(* Logix 5000 project; controller cal1632 1756-L62 rev 16.20; software revision 16.05; part 55 of 61 *)
(* tags used below, declared in another part *)
   p29_param_tension_hi_limit : REAL;   // Parameter Tension High Limit
   p29r16_drive_ok : BOOL;   // Winder B Drive Enable E-Stop Clear and Own Drive Healthy
   param_pos_db : REAL;   // C: Turret Position Dead Band
   pb_jog_turret_rev : BOOL;   // HMI PB: Jog Turret Rev
   turret_in_wda_run_position : BOOL;   // Turret In Winder A Run Position
   turret_in_wdb_run_position : BOOL;   // Turret In Winder B Run Position
   turret_index_permissive : BOOL;   // Turret Index Permissive No Turret Drive Fault AND Neither Winder Requesting Run
   wb_run_position : REAL;   // Turret Winder B Run Position
   wb_run_position_high_limit : REAL;
   wb_run_position_low_limit : REAL;
   winder_accel_rate : REAL;
   winder_decel_rate : REAL;
   AFI : BOOL;
   FAULT : BOOL;
   p00_wac : Accumulator;   // Winder Accumulator
   p00_wac_position_pct : REAL;   // Winder Accumulator Carriage Position Filtered [% of Stroke]
   p01_recipe_active : recipe;
   p01r02_plc_scan_time_in_sec : REAL;
   p01r09 : routine;
   p01r09_pb_global_reset : BOOL;
   p01r09_request_line_jog : BOOL;
   p01r13_line_running : BOOL;
   p01r13_line_slow_ramp : BOOL;
   p01r13_permissive_drives : BOOL;
   p02_real_from_hmi : hmi_real;
   p25_ao_selected_speed : REAL;
   p25r09_mode_thread : BOOL;
   p25r09_pb_jog_fwd : BOOL;
   p25r09_pb_jog_rev : BOOL;
   p29_ai_wb_torque : REAL;
   p29_ai_wdr_lc : REAL;
   p29_ao_wdrb_selected_speed : REAL;
   p29_di_wa_brake : BOOL;
   p29_di_wa_motor : BOOL;
   p29_di_wb_brake : BOOL;
   p29_di_wb_motor : BOOL;
   p29_di_wdr_b_start : BOOL;
   p29_di_wdr_b_stop : BOOL;
   p29_di_wdr_index_fwd : BOOL;
   p29_di_wdr_jog : BOOL;
   p29_param_payout_torque : REAL;   // Winder Torque Limit During Accumulator Payout Line Running [%]
   p29_param_soak : REAL;
   p29_param_start_speed_factor : REAL;   // Winder Start Speed Fraction of Line Speed Before Tension is Established Shared by Winder A and B
   p29_param_tension_ok_band : REAL;   // Winder Tension Established Band Shared by Winder A and B [lbf]
   p29_param_wind_out_speed : REAL;   // Winder Wind Out Speed Winder Speed with the Line Stopped Empties the Accumulator [fpm]
   p29_param_wind_out_stop_pct : REAL;   // Winder Wind Out Stop When the Accumulator Reaches This Position [% of Stroke]
   p29_param_wind_out_torque : REAL;   // Winder Torque Limit During Wind Out Line Stopped [%]
   p29_param_winder_accel_rate : REAL;   // Winder Common Speed Ramp Default Accel Rate Applied Only if winder_accel_rate is Zero
   p29_param_winder_decel_rate : REAL;   // Winder Common Speed Ramp Default Decel Rate Applied Only if winder_decel_rate is Zero
   p29_param_winder_jog_speed : REAL;
   p29_wda_status_word : INT;
   p29_wda_vfd : ABB_PROTOCOL_VFD;
   p29_wdb_control_word : INT;
   p29_wdb_status_word : INT;
   p29_wdb_vfd : ABB_PROTOCOL_VFD;
   p29r01 : routine;
   p29r02_tension_dev_max : REAL;
   p29r02_tension_dev_min : REAL;
   p29r02_wb_calc_torque_ref : REAL;
   p29r09_torque_mode : BOOL;
   p29r09_winder_b_active : BOOL;
   p29r11_index_active : BOOL;
   p29r11_speed_offset : REAL;
   p29r15 : routine;
   p29r15_request_run : BOOL;
   p29r15_run_permissive : BOOL;
   p29r15_timer_fault : TIMER[10];
   p29r15_timer_warning : TIMER[4];
   p29r15_wdra_active : BOOL;
   p29r16 : routine;
   p29r16_accel_rate : REAL;
   p29r16_acel_decel_ramp : SYS_ACC_DEC_RAMP;   // Winder B Speed Setpoint Ramp
   p29r16_ao_torque : REAL;
   p29r16_const_torque_ref : REAL;
   p29r16_decel_rate : REAL;
   p29r16_fast_accel_rate : REAL;
   p29r16_fast_decel_rate : REAL;
   p29r16_index_start_torque : REAL;
   p29r16_jog_torque_ref : REAL;
   p29r16_ramped_setpoint : REAL;   // Winder B Ramped Speed Setpoint [fpm]
   p29r16_request_jog_fwd : BOOL;
   p29r16_request_run : BOOL;
   p29r16_request_thread_fwd : BOOL;
   p29r16_request_thread_rev : BOOL;
   p29r16_run_permissive : BOOL;
   p29r16_selected_speed : REAL;
   p29r16_selected_torque : REAL;
   p29r16_soak_active : BOOL;
   p29r16_speed_factor : REAL;   // Winder B Speed Factor Multiplier on the Ramped Setpoint
   p29r16_speed_setpoint : REAL;   // Winder B Speed Setpoint [fpm]
   p29r16_state : DINT;
   p29r16_stop_dwell : TIMER;   // Winder B Stop Dwell Holds the winder after the stop PB so the nip closes first
   p29r16_tension_ok : BOOL;
   p29r16_thread_torque_ref : REAL;
   p29r16_timer_fault : TIMER[10];
   p29r16_timer_warning : TIMER[4];
   p29r16_torque_acc_rate : REAL;
   p29r16_torque_boost_acc_rate : REAL;
   p29r16_torque_boost_dec_rate : REAL;
   p29r16_torque_boost_ref : REAL;
   p29r16_torque_boost_timer : TIMER;
   p29r16_torque_dec_rate : REAL;
   p29r16_torque_fast_acc_rate : REAL;
   p29r16_torque_fast_dec_rate : REAL;
   p29r16_torque_high_ref : REAL;
   p29r16_torque_low_ref : REAL;
   p29r16_torque_mode_acc_rate : REAL;
   p29r16_torque_mode_dec_rate : REAL;
   p29r16_torque_ramp : SYS_ACC_DEC_RAMP;
   p29r16_torque_soak_acc_rate : REAL;
   p29r16_torque_soak_dec_rate : REAL;
   p29r16_torque_start_timer : TIMER;
   p29r16_vfd_start_request : BOOL;
   p29r16_wdrb_accel_decel : SYS_ACC_DEC_RAMP;
   p29r16_wdrb_active : BOOL;
   p29r16_wdrb_ramped_speed : REAL;
   p29r16_zero_speed : BOOL;
   p29r20 : routine;
(* P29_Winder, continued *)

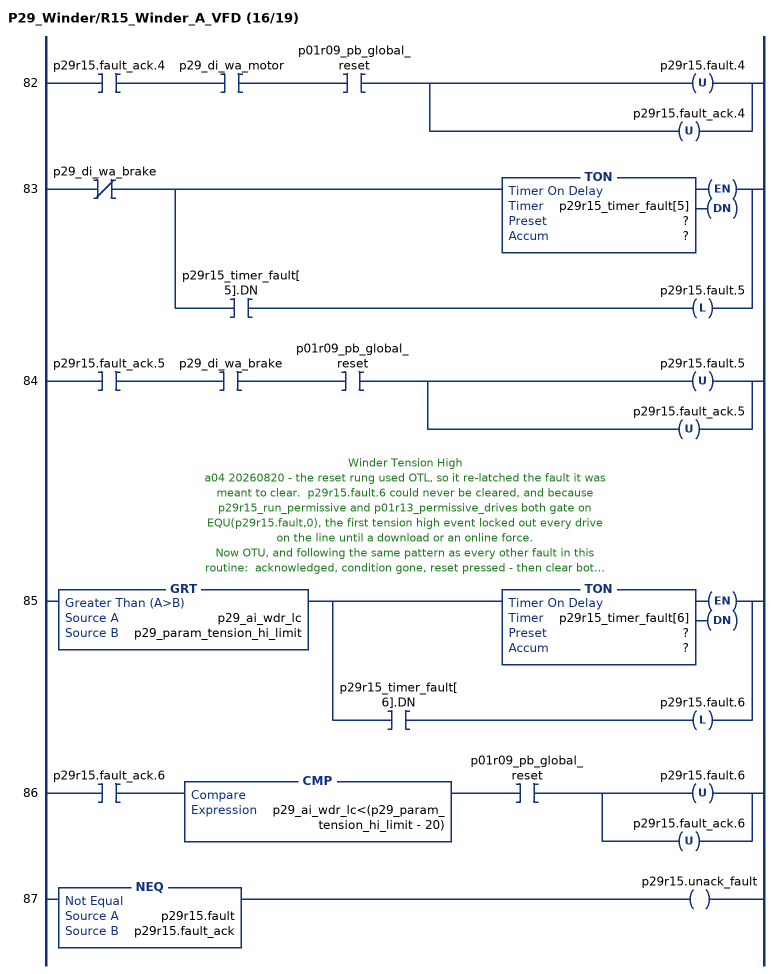
   [picture p1114: P29_Winder/R15_Winder_A_VFD rungs 82-87]
   82: XIC(p29r15.fault_ack.4)XIC(p29_di_wa_motor)XIC(p01r09_pb_global_reset)[OTU(p29r15.fault.4) ,OTU(p29r15.fault_ack.4) ];
   83: XIO(p29_di_wa_brake)[TON(p29r15_timer_fault[5],?,?) ,XIC(p29r15_timer_fault[5].DN) OTL(p29r15.fault.5) ];
   84: XIC(p29r15.fault_ack.5)XIC(p29_di_wa_brake)XIC(p01r09_pb_global_reset)[OTU(p29r15.fault.5) ,OTU(p29r15.fault_ack.5) ];
   // Winder Tension High
   // a04 20260820 - the reset rung used OTL, so it re-latched the fault it was
   // meant to clear.  p29r15.fault.6 could never be cleared, and because
   // p29r15_run_permissive and p01r13_permissive_drives both gate on
   // EQU(p29r15.fault,0), the first tension high event locked out every drive
   // on the line until a download or an online force.
   // Now OTU, and following the same pattern as every other fault in this
   // routine:  acknowledged, condition gone, reset pressed - then clear both
   // the fault bit and its ack bit so unack_fault clears with it.
   // Note p29_ai_wdr_lc is a single load cell shared by both winders, so a
   // tension excursion latches fault.6 on A and B together.  That is correct
   // for one web, but both need the reset.
   85: GRT(p29_ai_wdr_lc,p29_param_tension_hi_limit)[TON(p29r15_timer_fault[6],?,?) ,XIC(p29r15_timer_fault[6].DN) OTL(p29r15.fault.6) ];
   86: XIC(p29r15.fault_ack.6)CMP(p29_ai_wdr_lc<(p29_param_tension_hi_limit - 20))XIC(p01r09_pb_global_reset)[OTU(p29r15.fault.6) ,OTU(p29r15.fault_ack.6) ];
   87: NEQ(p29r15.fault,p29r15.fault_ack)OTE(p29r15.unack_fault);
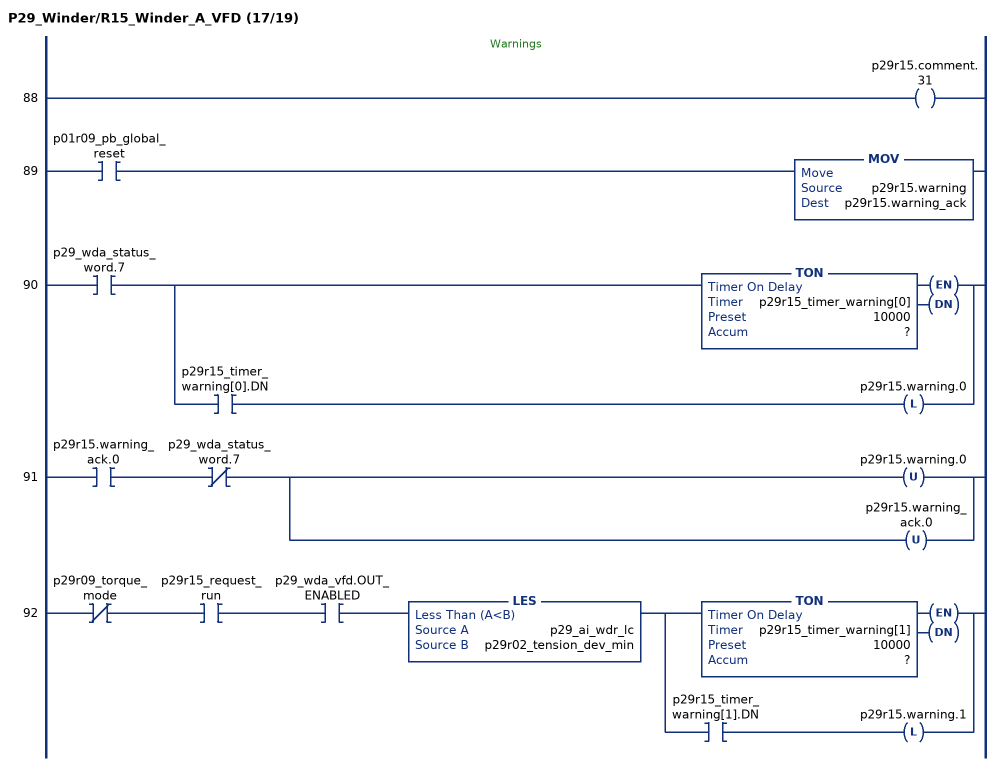
   // Warnings
   88: OTE(p29r15.comment.31);
   89: XIC(p01r09_pb_global_reset)MOV(p29r15.warning,p29r15.warning_ack);
   90: XIC(p29_wda_status_word.7)[TON(p29r15_timer_warning[0],?,?) ,XIC(p29r15_timer_warning[0].DN) OTL(p29r15.warning.0) ];
   91: XIC(p29r15.warning_ack.0)XIO(p29_wda_status_word.7)[OTU(p29r15.warning.0) ,OTU(p29r15.warning_ack.0) ];
   92: XIO(p29r09_torque_mode)XIC(p29r15_request_run)XIC(p29_wda_vfd.OUT_ENABLED)LES(p29_ai_wdr_lc,p29r02_tension_dev_min)[TON(p29r15_timer_warning[1],?,?) ,XIC(p29r15_timer_warning[1].DN) OTL(p29r15.warning.1) ];
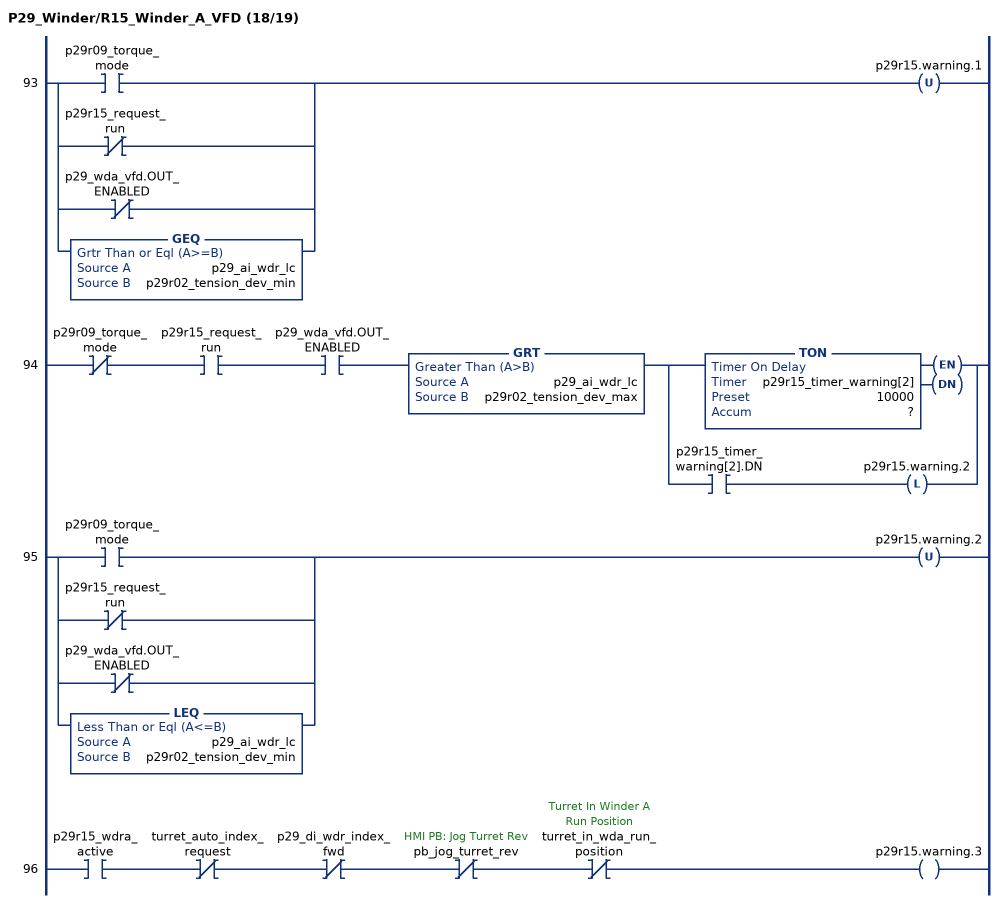
   93: [XIC(p29r09_torque_mode) ,XIO(p29r15_request_run) ,XIO(p29_wda_vfd.OUT_ENABLED) ,GEQ(p29_ai_wdr_lc,p29r02_tension_dev_min) ]OTU(p29r15.warning.1);
   94: XIO(p29r09_torque_mode)XIC(p29r15_request_run)XIC(p29_wda_vfd.OUT_ENABLED)GRT(p29_ai_wdr_lc,p29r02_tension_dev_max)[TON(p29r15_timer_warning[2],?,?) ,XIC(p29r15_timer_warning[2].DN) OTL(p29r15.warning.2) ];
   95: [XIC(p29r09_torque_mode) ,XIO(p29r15_request_run) ,XIO(p29_wda_vfd.OUT_ENABLED) ,LEQ(p29_ai_wdr_lc,p29r02_tension_dev_min) ]OTU(p29r15.warning.2);
   96: XIC(p29r15_wdra_active)XIO(turret_auto_index_request)XIO(p29_di_wdr_index_fwd)XIO(pb_jog_turret_rev)XIO(turret_in_wda_run_position)OTE(p29r15.warning.3);
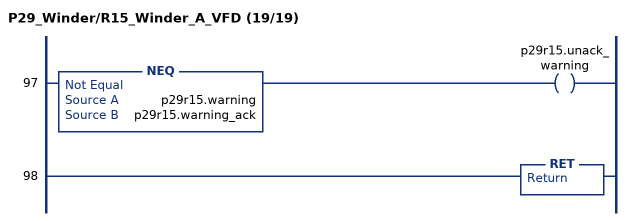
   97: NEQ(p29r15.warning,p29r15.warning_ack)OTE(p29r15.unack_warning);
   98: RET();
END_ROUTINE

ROUTINE R16_Winder_B_VFD   (* ladder *)
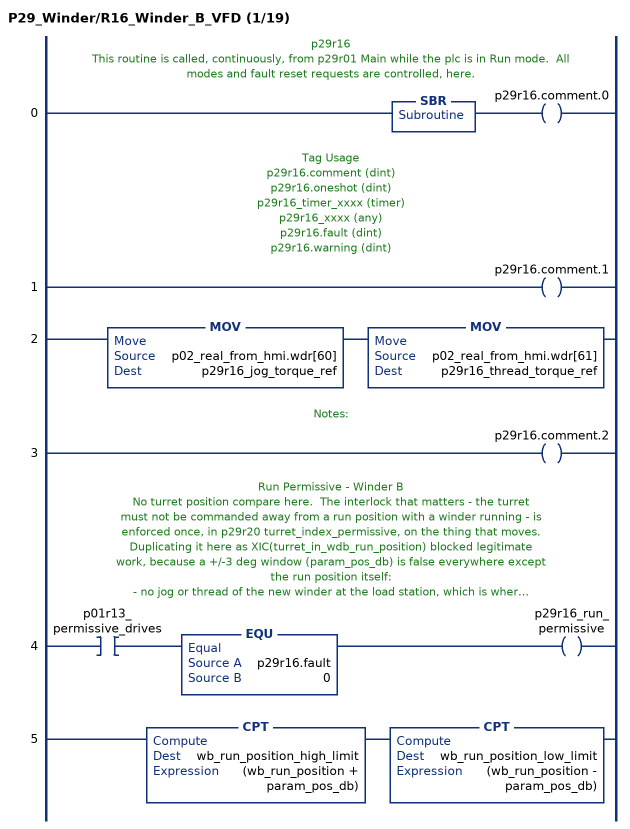
   // p29r16
   // This routine is called, continuously, from p29r01 Main while the plc is in Run mode.  All modes and fault reset requests are controlled, here.
   0: SBR()OTE(p29r16.comment.0);
   // Tag Usage
   // p29r16.comment (dint)
   // p29r16.oneshot (dint)
   // p29r16_timer_xxxx (timer)
   // p29r16_xxxx (any)
   // p29r16.fault (dint)
   // p29r16.warning (dint)
   1: OTE(p29r16.comment.1);
   2: MOV(p02_real_from_hmi.wdr[60],p29r16_jog_torque_ref)MOV(p02_real_from_hmi.wdr[61],p29r16_thread_torque_ref);
   // Notes:
   3: OTE(p29r16.comment.2);
   // Run Permissive - Winder B
   // No turret position compare here.  The interlock that matters - the turret
   // must not be commanded away from a run position with a winder running - is
   // enforced once, in p29r20 turret_index_permissive, on the thing that moves.
   // Duplicating it here as XIC(turret_in_wdb_run_position) blocked legitimate
   // work, because a +/-3 deg window (param_pos_db) is false everywhere except
   // the run position itself:
   //   - no jog or thread of the new winder at the load station, which is where
   //     the leader is attached and has to be wound on
   //   - no winding the tail off the doffed roll at doff position
   //   - no accumulator wind-out unless the turret happens to be at run
   //   - the winder dropped out 0.7 s into a doff index, web still tensioned
   // Rev 20260825 a23
   4: XIC(p01r13_permissive_drives)EQU(p29r16.fault,0)OTE(p29r16_run_permissive);
   5: CPT(wb_run_position_high_limit,(wb_run_position + param_pos_db))CPT(wb_run_position_low_limit,(wb_run_position - param_pos_db));
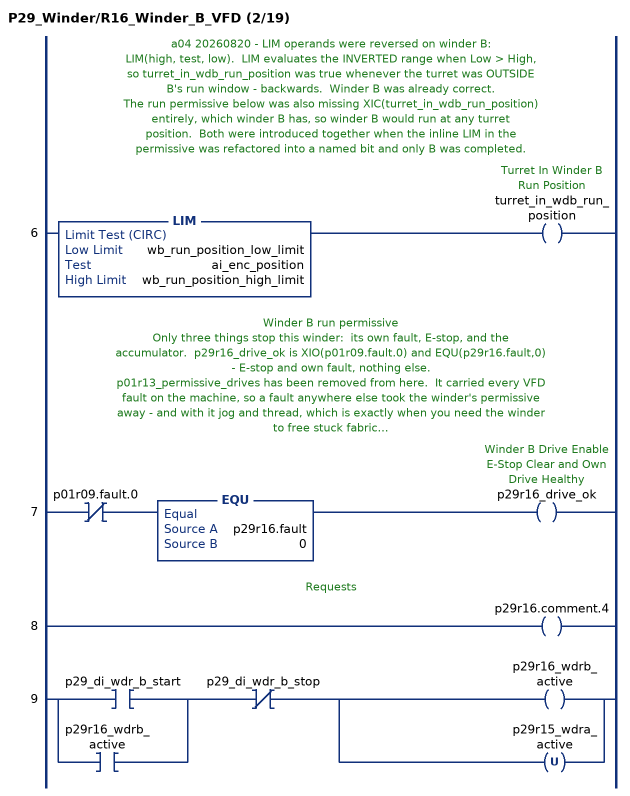
   // a04 20260820 - LIM operands were reversed on winder B:
   // LIM(high, test, low).  LIM evaluates the INVERTED range when Low > High,
   // so turret_in_wdb_run_position was true whenever the turret was OUTSIDE
   // B's run window - backwards.  Winder B was already correct.
   // The run permissive below was also missing XIC(turret_in_wdb_run_position)
   // entirely, which winder B has, so winder B would run at any turret
   // position.  Both were introduced together when the inline LIM in the
   // permissive was refactored into a named bit and only B was completed.
   6: LIM(wb_run_position_low_limit,ai_enc_position,wb_run_position_high_limit)OTE(turret_in_wdb_run_position);
   // Winder B run permissive
   // Only three things stop this winder:  its own fault, E-stop, and the
   // accumulator.  p29r16_drive_ok is XIO(p01r09.fault.0) and EQU(p29r16.fault,0)
   // - E-stop and own fault, nothing else.
   // p01r13_permissive_drives has been removed from here.  It carried every VFD
   // fault on the machine, so a fault anywhere else took the winder's permissive
   // away - and with it jog and thread, which is exactly when you need the winder
   // to free stuck fabric.
   // The turret window stays:  the winder must not run with the turret away from
   // its run position.  The accumulator has its say through the run request and
   // through wac_empty_stop / wac_full_stop on the line.
   // Rev 20260825 a16
   7: XIO(p01r09.fault.0)EQU(p29r16.fault,0)OTE(p29r16_drive_ok);
   // Requests
   8: OTE(p29r16.comment.4);
   9: [XIC(p29_di_wdr_b_start) ,XIC(p29r16_wdrb_active) ]XIO(p29_di_wdr_b_stop)[OTE(p29r16_wdrb_active) ,OTU(p29r15_wdra_active) ];
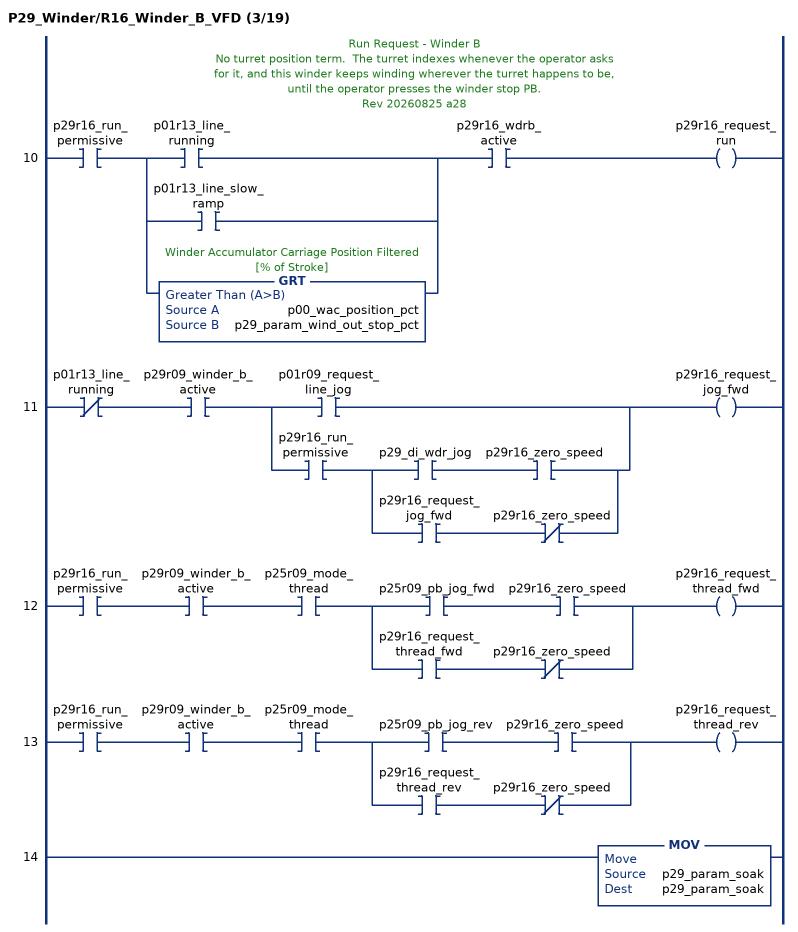
   // Run Request - Winder B
   // No turret position term.  The turret indexes whenever the operator asks
   // for it, and this winder keeps winding wherever the turret happens to be,
   // until the operator presses the winder stop PB.
   // Rev 20260825 a28
   10: XIC(p29r16_run_permissive)[XIC(p01r13_line_running) ,XIC(p01r13_line_slow_ramp) ,GRT(p00_wac_position_pct,p29_param_wind_out_stop_pct) ]XIC(p29r16_wdrb_active)OTE(p29r16_request_run);
   11: XIO(p01r13_line_running)XIC(p29r09_winder_b_active)[XIC(p01r09_request_line_jog) ,XIC(p29r16_run_permissive) [XIC(p29_di_wdr_jog) XIC(p29r16_zero_speed) ,XIC(p29r16_request_jog_fwd) XIO(p29r16_zero_speed) ] ]OTE(p29r16_request_jog_fwd);
   12: XIC(p29r16_run_permissive)XIC(p29r09_winder_b_active)XIC(p25r09_mode_thread)[XIC(p25r09_pb_jog_fwd) XIC(p29r16_zero_speed) ,XIC(p29r16_request_thread_fwd) XIO(p29r16_zero_speed) ]OTE(p29r16_request_thread_fwd);
   13: XIC(p29r16_run_permissive)XIC(p29r09_winder_b_active)XIC(p25r09_mode_thread)[XIC(p25r09_pb_jog_rev) XIC(p29r16_zero_speed) ,XIC(p29r16_request_thread_rev) XIO(p29r16_zero_speed) ]OTE(p29r16_request_thread_rev);
   14: MOV(p29_param_soak,p29_param_soak);
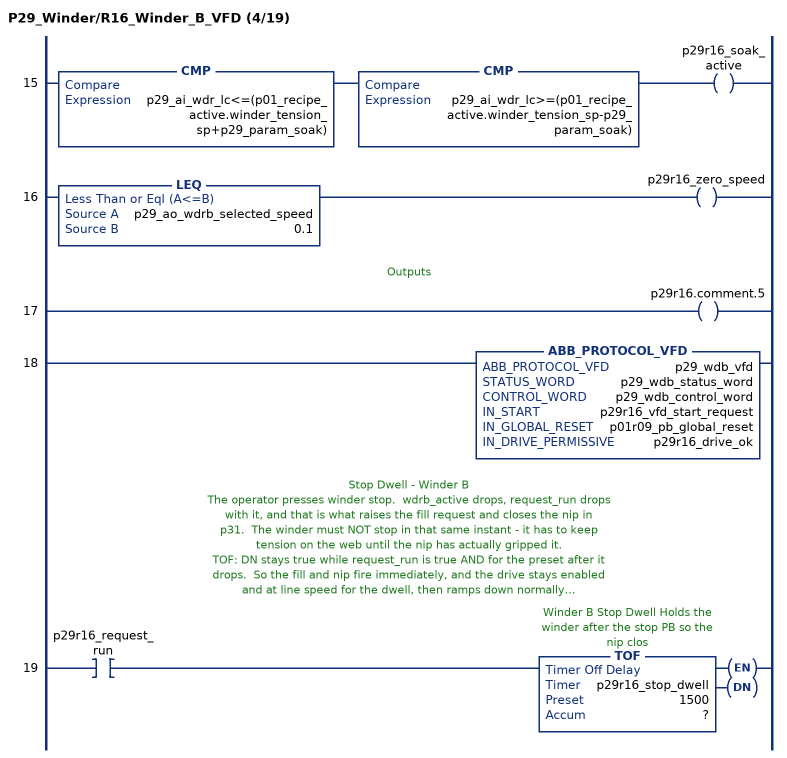
   15: CMP(p29_ai_wdr_lc<=(p01_recipe_active.winder_tension_sp+p29_param_soak))CMP(p29_ai_wdr_lc>=(p01_recipe_active.winder_tension_sp-p29_param_soak))OTE(p29r16_soak_active);
   16: LEQ(p29_ao_wdrb_selected_speed,0.1)OTE(p29r16_zero_speed);
   // Outputs
   17: OTE(p29r16.comment.5);
   18: ABB_PROTOCOL_VFD(p29_wdb_vfd,p29_wdb_status_word,p29_wdb_control_word,p29r16_vfd_start_request,p01r09_pb_global_reset,p29r16_drive_ok);
   // Stop Dwell - Winder B
   // The operator presses winder stop.  wdrb_active drops, request_run drops
   // with it, and that is what raises the fill request and closes the nip in
   // p31.  The winder must NOT stop in that same instant - it has to keep
   // tension on the web until the nip has actually gripped it.
   // TOF: DN stays true while request_run is true AND for the preset after it
   // drops.  So the fill and nip fire immediately, and the drive stays enabled
   // and at line speed for the dwell, then ramps down normally.
   // Rev 20260825 a30
   19: XIC(p29r16_request_run)TOF(p29r16_stop_dwell,?,?);
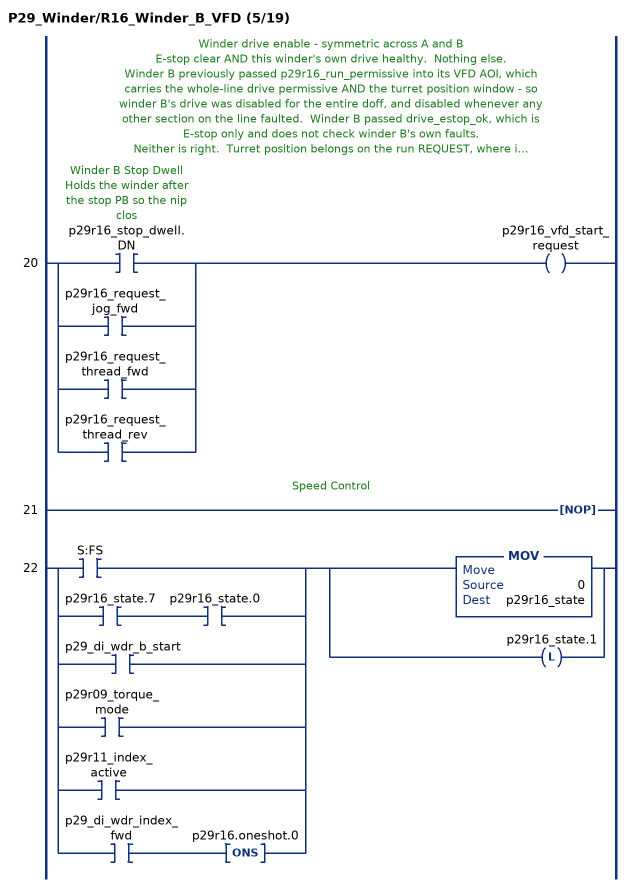
   // Winder drive enable - symmetric across A and B
   // E-stop clear AND this winder's own drive healthy.  Nothing else.
   // Winder B previously passed p29r16_run_permissive into its VFD AOI, which
   // carries the whole-line drive permissive AND the turret position window - so
   // winder B's drive was disabled for the entire doff, and disabled whenever any
   // other section on the line faulted.  Winder B passed drive_estop_ok, which is
   // E-stop only and does not check winder B's own faults.
   // Neither is right.  Turret position belongs on the run REQUEST, where it
   // already is, not on the drive enable; and the whole-line permissive would
   // stop you jogging a winder to free the fabric while another section is down.
   // Own-drive faults do belong here.
   // Rev 20260825 a12
   20: [XIC(p29r16_stop_dwell.DN) ,XIC(p29r16_request_jog_fwd) ,XIC(p29r16_request_thread_fwd) ,XIC(p29r16_request_thread_rev) ]OTE(p29r16_vfd_start_request);
   // Speed Control
   21: NOP();
   22: [XIC(S:FS) ,XIC(p29r16_state.7) XIC(p29r16_state.0) ,XIC(p29_di_wdr_b_start) ,XIC(p29r09_torque_mode) ,XIC(p29r11_index_active) ,XIC(p29_di_wdr_index_fwd) ONS(p29r16.oneshot.0) ][MOV(0,p29r16_state) ,OTL(p29r16_state.1) ];
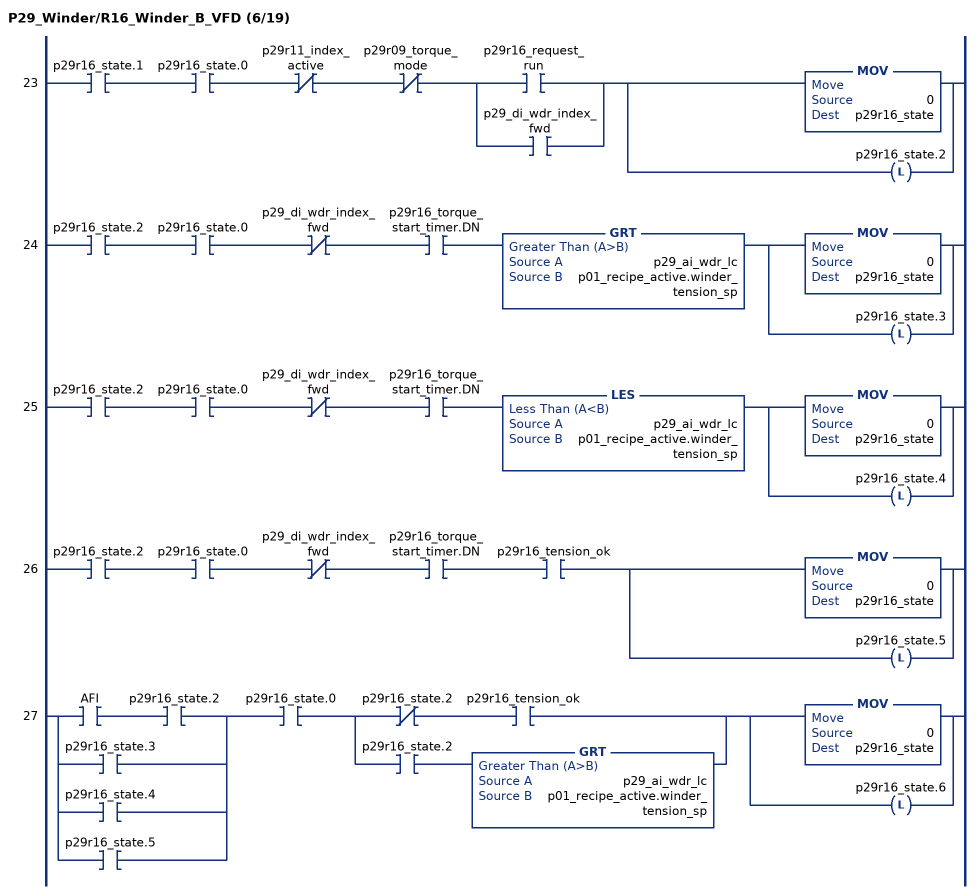
   23: XIC(p29r16_state.1)XIC(p29r16_state.0)XIO(p29r11_index_active)XIO(p29r09_torque_mode)[XIC(p29r16_request_run) ,XIC(p29_di_wdr_index_fwd) ][MOV(0,p29r16_state) ,OTL(p29r16_state.2) ];
   24: XIC(p29r16_state.2)XIC(p29r16_state.0)XIO(p29_di_wdr_index_fwd)XIC(p29r16_torque_start_timer.DN)GRT(p29_ai_wdr_lc,p01_recipe_active.winder_tension_sp)[MOV(0,p29r16_state) ,OTL(p29r16_state.3) ];
   25: XIC(p29r16_state.2)XIC(p29r16_state.0)XIO(p29_di_wdr_index_fwd)XIC(p29r16_torque_start_timer.DN)LES(p29_ai_wdr_lc,p01_recipe_active.winder_tension_sp)[MOV(0,p29r16_state) ,OTL(p29r16_state.4) ];
   26: XIC(p29r16_state.2)XIC(p29r16_state.0)XIO(p29_di_wdr_index_fwd)XIC(p29r16_torque_start_timer.DN)XIC(p29r16_tension_ok)[MOV(0,p29r16_state) ,OTL(p29r16_state.5) ];
   27: [XIC(AFI) XIC(p29r16_state.2) ,XIC(p29r16_state.3) ,XIC(p29r16_state.4) ,XIC(p29r16_state.5) ]XIC(p29r16_state.0)[XIO(p29r16_state.2) XIC(p29r16_tension_ok) ,XIC(p29r16_state.2) GRT(p29_ai_wdr_lc,p01_recipe_active.winder_tension_sp) ][MOV(0,p29r16_state) ,OTL(p29r16_state.6) ];
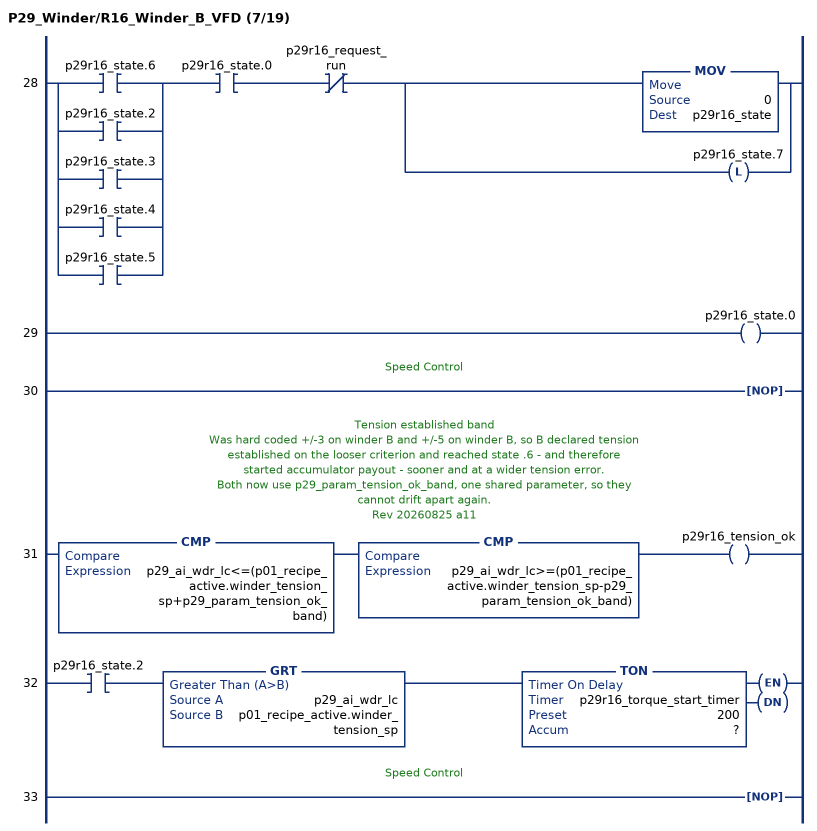
   28: [XIC(p29r16_state.6) ,XIC(p29r16_state.2) ,XIC(p29r16_state.3) ,XIC(p29r16_state.4) ,XIC(p29r16_state.5) ]XIC(p29r16_state.0)XIO(p29r16_request_run)[MOV(0,p29r16_state) ,OTL(p29r16_state.7) ];
   29: OTE(p29r16_state.0);
   // Speed Control
   30: NOP();
   // Tension established band
   // Was hard coded +/-3 on winder B and +/-5 on winder B, so B declared tension
   // established on the looser criterion and reached state .6 - and therefore
   // started accumulator payout - sooner and at a wider tension error.
   // Both now use p29_param_tension_ok_band, one shared parameter, so they
   // cannot drift apart again.
   // Rev 20260825 a11
   31: CMP(p29_ai_wdr_lc<=(p01_recipe_active.winder_tension_sp+p29_param_tension_ok_band))CMP(p29_ai_wdr_lc>=(p01_recipe_active.winder_tension_sp-p29_param_tension_ok_band))OTE(p29r16_tension_ok);
   32: XIC(p29r16_state.2)GRT(p29_ai_wdr_lc,p01_recipe_active.winder_tension_sp)TON(p29r16_torque_start_timer,?,?);
   // Speed Control
   33: NOP();
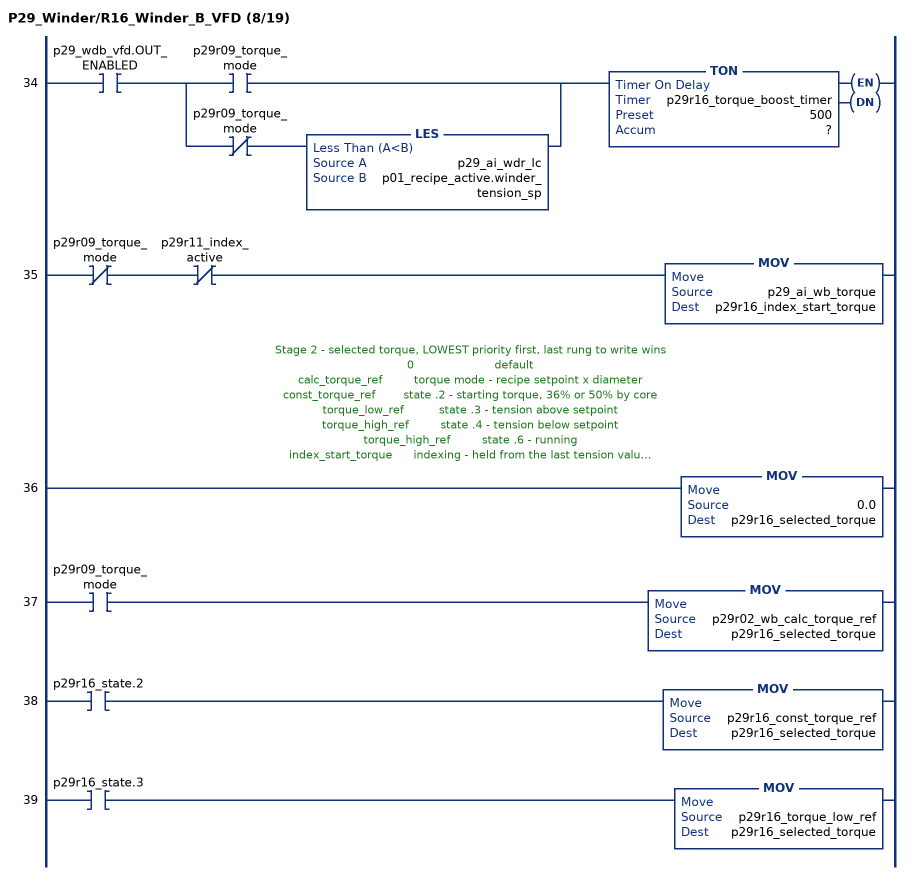
   34: XIC(p29_wdb_vfd.OUT_ENABLED)[XIC(p29r09_torque_mode) ,XIO(p29r09_torque_mode) LES(p29_ai_wdr_lc,p01_recipe_active.winder_tension_sp) ]TON(p29r16_torque_boost_timer,?,?);
   35: XIO(p29r09_torque_mode)XIO(p29r11_index_active)MOV(p29_ai_wb_torque,p29r16_index_start_torque);
   // Stage 2 - selected torque, LOWEST priority first, last rung to write wins
   //    0                       default
   //    calc_torque_ref         torque mode - recipe setpoint x diameter
   //    const_torque_ref        state .2 - starting torque, 36% or 50% by core
   //    torque_low_ref          state .3 - tension above setpoint
   //    torque_high_ref         state .4 - tension below setpoint
   //    torque_high_ref         state .6 - running
   //    index_start_torque      indexing - held from the last tension value
   //    jog_torque_ref          jog
   //    thread_torque_ref       thread
   //    torque_boost_ref        boost timer or start pushbutton
   //    payout_torque           accumulator paying out, line running
   //    wind_out_torque         accumulator paying out, line stopped
   36: MOV(0.0,p29r16_selected_torque);
   37: XIC(p29r09_torque_mode)MOV(p29r02_wb_calc_torque_ref,p29r16_selected_torque);
   38: XIC(p29r16_state.2)MOV(p29r16_const_torque_ref,p29r16_selected_torque);
   39: XIC(p29r16_state.3)MOV(p29r16_torque_low_ref,p29r16_selected_torque);
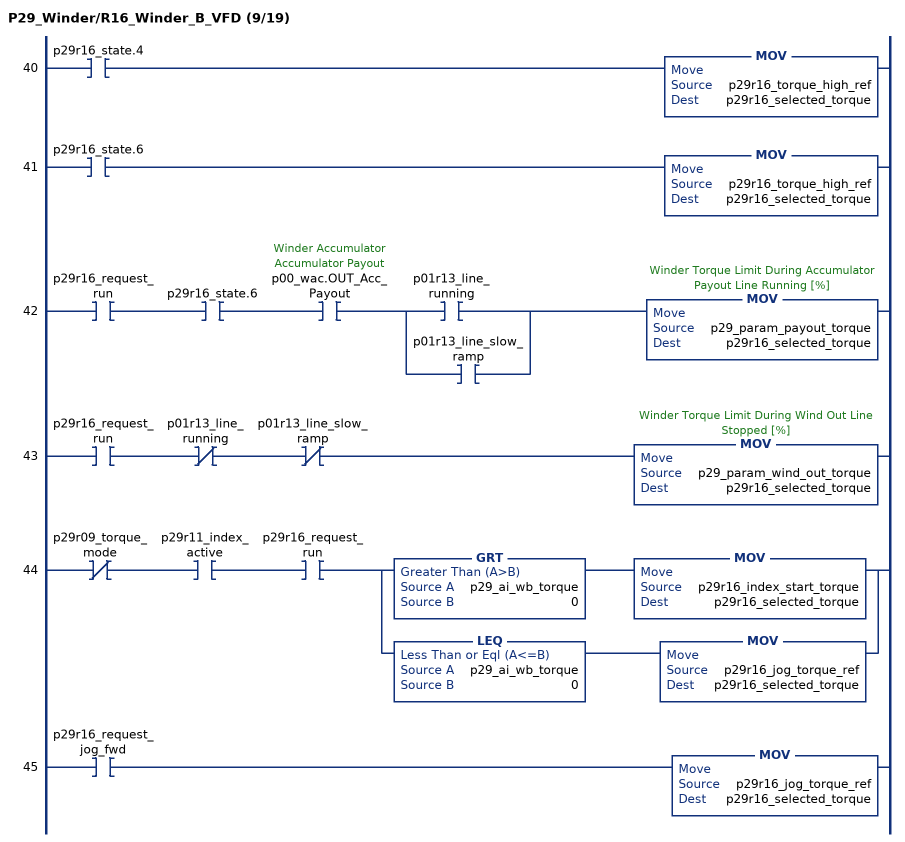
   40: XIC(p29r16_state.4)MOV(p29r16_torque_high_ref,p29r16_selected_torque);
   41: XIC(p29r16_state.6)MOV(p29r16_torque_high_ref,p29r16_selected_torque);
   42: XIC(p29r16_request_run)XIC(p29r16_state.6)XIC(p00_wac.OUT_Acc_Payout)[XIC(p01r13_line_running) ,XIC(p01r13_line_slow_ramp) ]MOV(p29_param_payout_torque,p29r16_selected_torque);
   43: XIC(p29r16_request_run)XIO(p01r13_line_running)XIO(p01r13_line_slow_ramp)MOV(p29_param_wind_out_torque,p29r16_selected_torque);
   44: XIO(p29r09_torque_mode)XIC(p29r11_index_active)XIC(p29r16_request_run)[GRT(p29_ai_wb_torque,0) MOV(p29r16_index_start_torque,p29r16_selected_torque) ,LEQ(p29_ai_wb_torque,0) MOV(p29r16_jog_torque_ref,p29r16_selected_torque) ];
   45: XIC(p29r16_request_jog_fwd)MOV(p29r16_jog_torque_ref,p29r16_selected_torque);
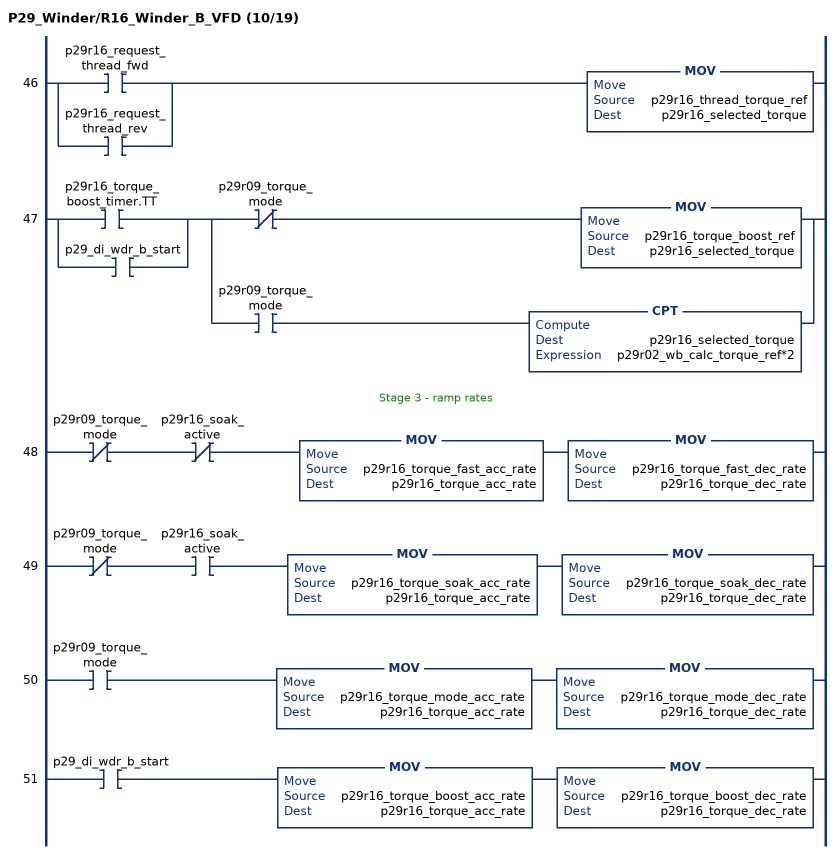
   46: [XIC(p29r16_request_thread_fwd) ,XIC(p29r16_request_thread_rev) ]MOV(p29r16_thread_torque_ref,p29r16_selected_torque);
   47: [XIC(p29r16_torque_boost_timer.TT) ,XIC(p29_di_wdr_b_start) ][XIO(p29r09_torque_mode) MOV(p29r16_torque_boost_ref,p29r16_selected_torque) ,XIC(p29r09_torque_mode) CPT(p29r16_selected_torque,p29r02_wb_calc_torque_ref*2) ];
   // Stage 3 - ramp rates
   48: XIO(p29r09_torque_mode)XIO(p29r16_soak_active)MOV(p29r16_torque_fast_acc_rate,p29r16_torque_acc_rate)MOV(p29r16_torque_fast_dec_rate,p29r16_torque_dec_rate);
   49: XIO(p29r09_torque_mode)XIC(p29r16_soak_active)MOV(p29r16_torque_soak_acc_rate,p29r16_torque_acc_rate)MOV(p29r16_torque_soak_dec_rate,p29r16_torque_dec_rate);
   50: XIC(p29r09_torque_mode)MOV(p29r16_torque_mode_acc_rate,p29r16_torque_acc_rate)MOV(p29r16_torque_mode_dec_rate,p29r16_torque_dec_rate);
   51: XIC(p29_di_wdr_b_start)MOV(p29r16_torque_boost_acc_rate,p29r16_torque_acc_rate)MOV(p29r16_torque_boost_dec_rate,p29r16_torque_dec_rate);
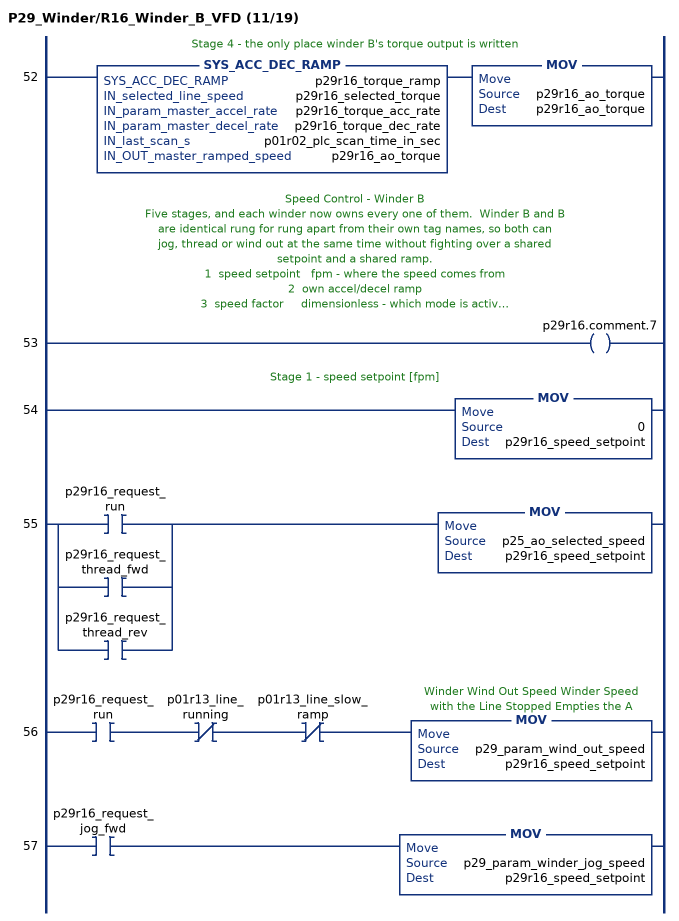
   // Stage 4 - the only place winder B's torque output is written
   52: SYS_ACC_DEC_RAMP(p29r16_torque_ramp,p29r16_selected_torque,p29r16_torque_acc_rate,p29r16_torque_dec_rate,p01r02_plc_scan_time_in_sec,p29r16_ao_torque)MOV(p29r16_ao_torque,p29r16_ao_torque);
   // Speed Control - Winder B
   // Five stages, and each winder now owns every one of them.  Winder B and B
   // are identical rung for rung apart from their own tag names, so both can
   // jog, thread or wind out at the same time without fighting over a shared
   // setpoint and a shared ramp.
   //   1  speed setpoint   fpm - where the speed comes from
   //   2  own accel/decel ramp
   //   3  speed factor     dimensionless - which mode is active
   //   4  one multiply     the ONLY place this winder's speed is calculated
   //   5  output ramp and clamp
   // This replaces a cascade of nine writes to p29r16_selected_speed and four to
   // a shared winder_speed_setpoint, where the last rung to execute won and the
   // precedence was nowhere stated.  Two faults came straight out of that:
   //   - the shared MOV(0,winder_speed_setpoint) fired whenever the line was not
   //     running and no jog was requested, which cancelled the wind out setpoint
   //     two rungs after it was written.  Wind out never ran.
   //   - the shared ramp lived inside p29r16, so it executed before p29r16 had
   //     written the setpoint at all.
   // Stage 3 is still a priority cascade - that is idiomatic in ladder - but it
   // is over a dimensionless factor, listed lowest priority first, and it is
   // trendable online so the active mode can be seen rather than inferred.
   // Rev 20260825 a18
   53: OTE(p29r16.comment.7);
   // Stage 1 - speed setpoint [fpm]
   54: MOV(0,p29r16_speed_setpoint);
   55: [XIC(p29r16_request_run) ,XIC(p29r16_request_thread_fwd) ,XIC(p29r16_request_thread_rev) ]MOV(p25_ao_selected_speed,p29r16_speed_setpoint);
   56: XIC(p29r16_request_run)XIO(p01r13_line_running)XIO(p01r13_line_slow_ramp)MOV(p29_param_wind_out_speed,p29r16_speed_setpoint);
   57: XIC(p29r16_request_jog_fwd)MOV(p29_param_winder_jog_speed,p29r16_speed_setpoint);
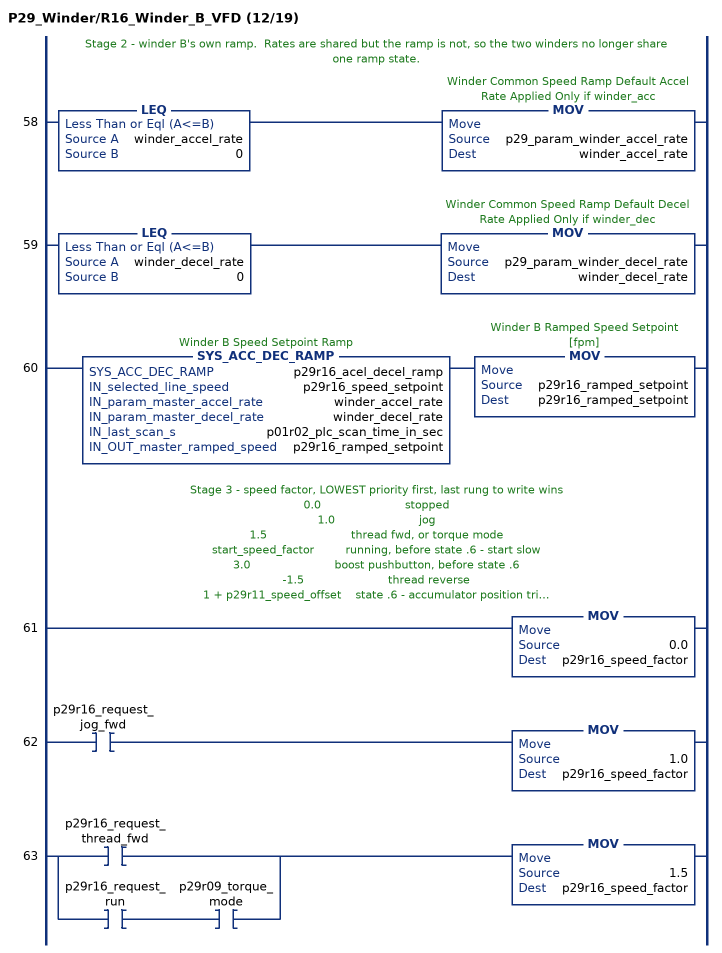
   // Stage 2 - winder B's own ramp.  Rates are shared but the ramp is not, so the two winders no longer share one ramp state.
   58: LEQ(winder_accel_rate,0)MOV(p29_param_winder_accel_rate,winder_accel_rate);
   59: LEQ(winder_decel_rate,0)MOV(p29_param_winder_decel_rate,winder_decel_rate);
   60: SYS_ACC_DEC_RAMP(p29r16_acel_decel_ramp,p29r16_speed_setpoint,winder_accel_rate,winder_decel_rate,p01r02_plc_scan_time_in_sec,p29r16_ramped_setpoint)MOV(p29r16_ramped_setpoint,p29r16_ramped_setpoint);
   // Stage 3 - speed factor, LOWEST priority first, last rung to write wins
   //    0.0                        stopped
   //    1.0                        jog
   //    1.5                        thread fwd, or torque mode
   //    start_speed_factor         running, before state .6 - start slow
   //    3.0                        boost pushbutton, before state .6
   //   -1.5                        thread reverse
   //    1 + p29r11_speed_offset    state .6 - accumulator position trim
   //    1.0                        line stopped - wind out, trim bypassed
   //    0.0                        turret going to doff
   61: MOV(0.0,p29r16_speed_factor);
   62: XIC(p29r16_request_jog_fwd)MOV(1.0,p29r16_speed_factor);
   63: [XIC(p29r16_request_thread_fwd) ,XIC(p29r16_request_run) XIC(p29r09_torque_mode) ]MOV(1.5,p29r16_speed_factor);
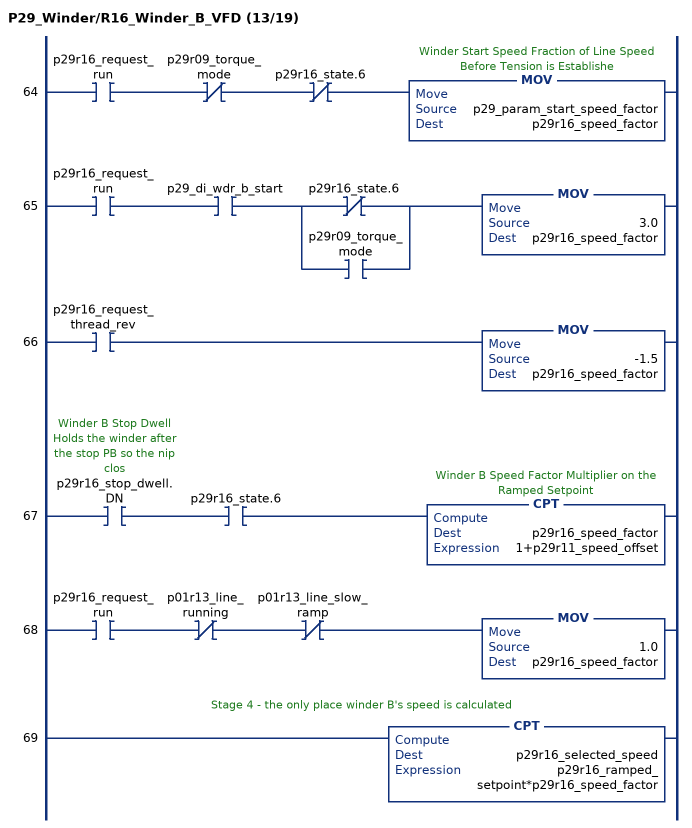
   64: XIC(p29r16_request_run)XIO(p29r09_torque_mode)XIO(p29r16_state.6)MOV(p29_param_start_speed_factor,p29r16_speed_factor);
   65: XIC(p29r16_request_run)XIC(p29_di_wdr_b_start)[XIO(p29r16_state.6) ,XIC(p29r09_torque_mode) ]MOV(3.0,p29r16_speed_factor);
   66: XIC(p29r16_request_thread_rev)MOV(-1.5,p29r16_speed_factor);
   67: XIC(p29r16_stop_dwell.DN)XIC(p29r16_state.6)CPT(p29r16_speed_factor,1+p29r11_speed_offset);
   68: XIC(p29r16_request_run)XIO(p01r13_line_running)XIO(p01r13_line_slow_ramp)MOV(1.0,p29r16_speed_factor);
   // Stage 4 - the only place winder B's speed is calculated
   69: CPT(p29r16_selected_speed,p29r16_ramped_setpoint*p29r16_speed_factor);
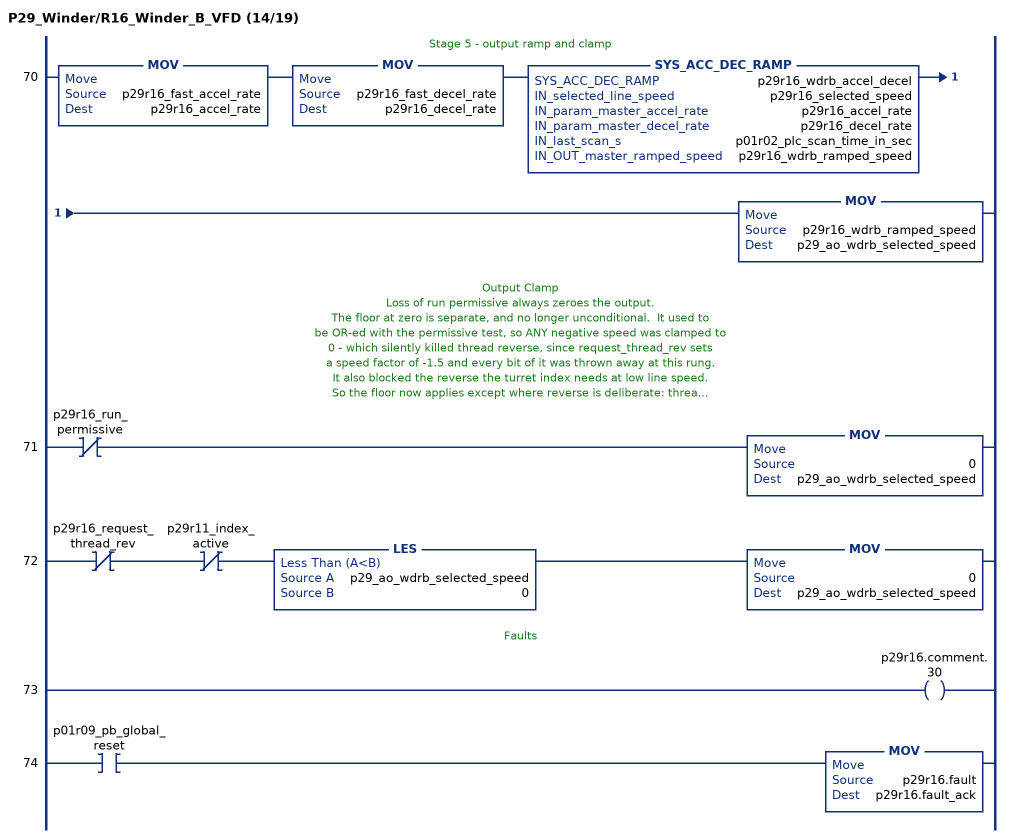
   // Stage 5 - output ramp and clamp
   70: MOV(p29r16_fast_accel_rate,p29r16_accel_rate)MOV(p29r16_fast_decel_rate,p29r16_decel_rate)SYS_ACC_DEC_RAMP(p29r16_wdrb_accel_decel,p29r16_selected_speed,p29r16_accel_rate,p29r16_decel_rate,p01r02_plc_scan_time_in_sec,p29r16_wdrb_ramped_speed)MOV(p29r16_wdrb_ramped_speed,p29_ao_wdrb_selected_speed);
   // Output Clamp
   // Loss of run permissive always zeroes the output.
   // The floor at zero is separate, and no longer unconditional.  It used to
   // be OR-ed with the permissive test, so ANY negative speed was clamped to
   // 0 - which silently killed thread reverse, since request_thread_rev sets
   // a speed factor of -1.5 and every bit of it was thrown away at this rung.
   // It also blocked the reverse the turret index needs at low line speed.
   // So the floor now applies except where reverse is deliberate: thread
   // reverse, or an index in progress.  SYS_SPEED_TO_VFD passes a negative
   // speed straight through - it only guards gear ratio and diameter - so the
   // drive must be configured for a bipolar speed reference for this to do
   // anything at the motor.
   // Rev 20260825 a26
   71: XIO(p29r16_run_permissive)MOV(0,p29_ao_wdrb_selected_speed);
   72: XIO(p29r16_request_thread_rev)XIO(p29r11_index_active)LES(p29_ao_wdrb_selected_speed,0)MOV(0,p29_ao_wdrb_selected_speed);
   // Faults
   73: OTE(p29r16.comment.30);
   74: XIC(p01r09_pb_global_reset)MOV(p29r16.fault,p29r16.fault_ack);
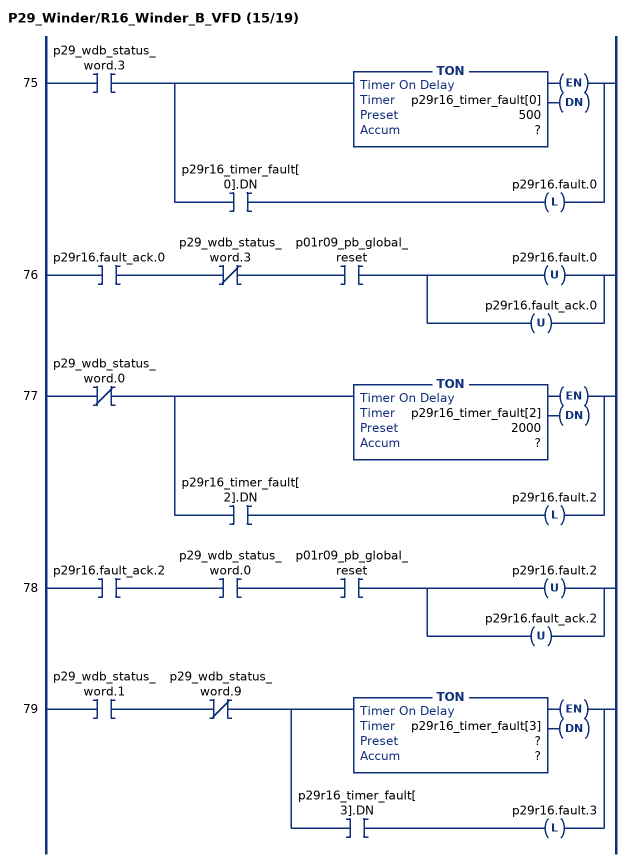
   75: XIC(p29_wdb_status_word.3)[TON(p29r16_timer_fault[0],?,?) ,XIC(p29r16_timer_fault[0].DN) OTL(p29r16.fault.0) ];
   76: XIC(p29r16.fault_ack.0)XIO(p29_wdb_status_word.3)XIC(p01r09_pb_global_reset)[OTU(p29r16.fault.0) ,OTU(p29r16.fault_ack.0) ];
   77: XIO(p29_wdb_status_word.0)[TON(p29r16_timer_fault[2],?,?) ,XIC(p29r16_timer_fault[2].DN) OTL(p29r16.fault.2) ];
   78: XIC(p29r16.fault_ack.2)XIC(p29_wdb_status_word.0)XIC(p01r09_pb_global_reset)[OTU(p29r16.fault.2) ,OTU(p29r16.fault_ack.2) ];
   79: XIC(p29_wdb_status_word.1)XIO(p29_wdb_status_word.9)[TON(p29r16_timer_fault[3],?,?) ,XIC(p29r16_timer_fault[3].DN) OTL(p29r16.fault.3) ];
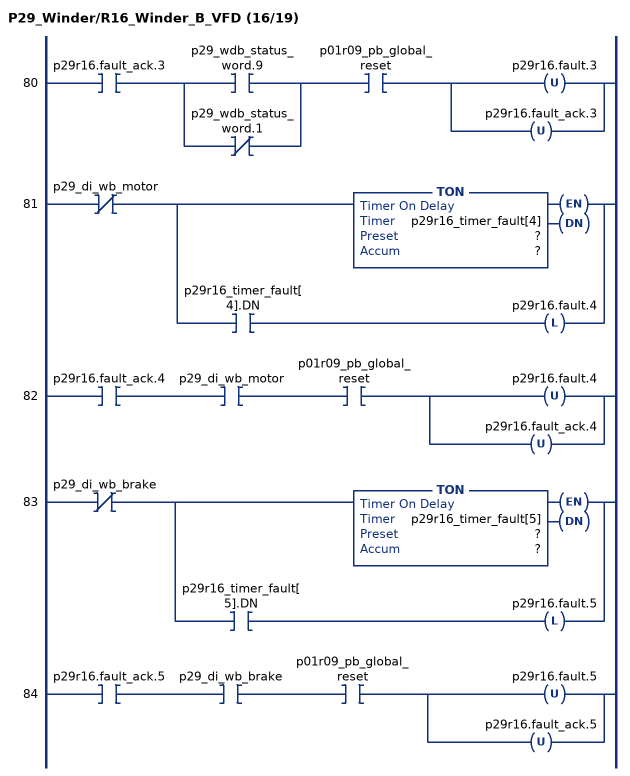
   80: XIC(p29r16.fault_ack.3)[XIC(p29_wdb_status_word.9) ,XIO(p29_wdb_status_word.1) ]XIC(p01r09_pb_global_reset)[OTU(p29r16.fault.3) ,OTU(p29r16.fault_ack.3) ];
   81: XIO(p29_di_wb_motor)[TON(p29r16_timer_fault[4],?,?) ,XIC(p29r16_timer_fault[4].DN) OTL(p29r16.fault.4) ];
   82: XIC(p29r16.fault_ack.4)XIC(p29_di_wb_motor)XIC(p01r09_pb_global_reset)[OTU(p29r16.fault.4) ,OTU(p29r16.fault_ack.4) ];
   83: XIO(p29_di_wb_brake)[TON(p29r16_timer_fault[5],?,?) ,XIC(p29r16_timer_fault[5].DN) OTL(p29r16.fault.5) ];
   84: XIC(p29r16.fault_ack.5)XIC(p29_di_wb_brake)XIC(p01r09_pb_global_reset)[OTU(p29r16.fault.5) ,OTU(p29r16.fault_ack.5) ];
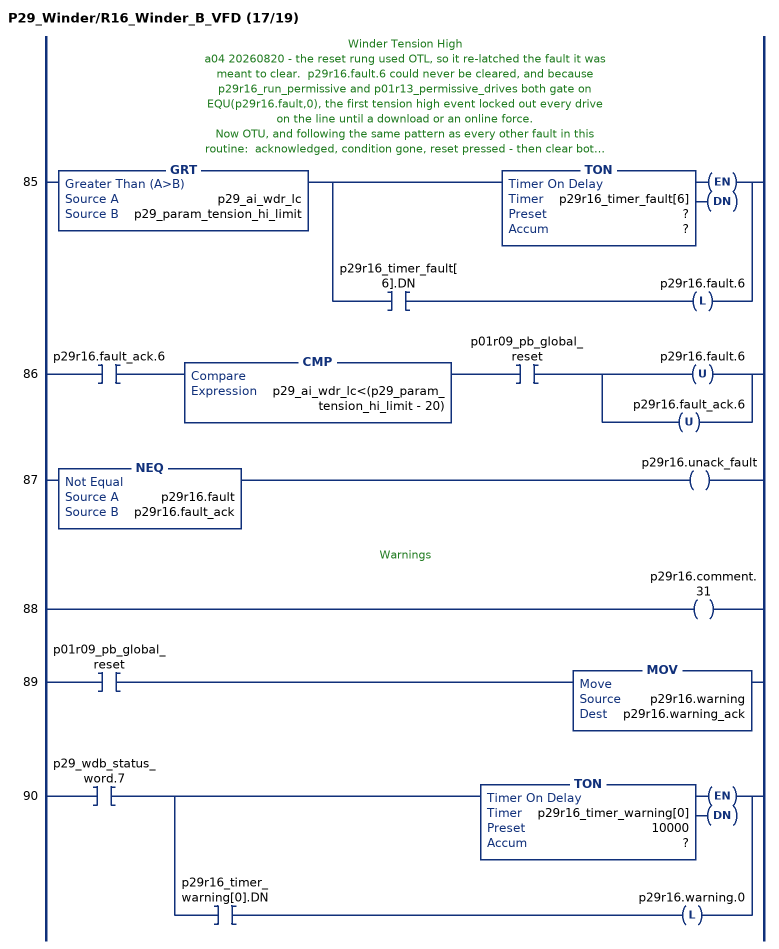
   // Winder Tension High
   // a04 20260820 - the reset rung used OTL, so it re-latched the fault it was
   // meant to clear.  p29r16.fault.6 could never be cleared, and because
   // p29r16_run_permissive and p01r13_permissive_drives both gate on
   // EQU(p29r16.fault,0), the first tension high event locked out every drive
   // on the line until a download or an online force.
   // Now OTU, and following the same pattern as every other fault in this
   // routine:  acknowledged, condition gone, reset pressed - then clear both
   // the fault bit and its ack bit so unack_fault clears with it.
   // Note p29_ai_wdr_lc is a single load cell shared by both winders, so a
   // tension excursion latches fault.6 on A and B together.  That is correct
   // for one web, but both need the reset.
   85: GRT(p29_ai_wdr_lc,p29_param_tension_hi_limit)[TON(p29r16_timer_fault[6],?,?) ,XIC(p29r16_timer_fault[6].DN) OTL(p29r16.fault.6) ];
   86: XIC(p29r16.fault_ack.6)CMP(p29_ai_wdr_lc<(p29_param_tension_hi_limit - 20))XIC(p01r09_pb_global_reset)[OTU(p29r16.fault.6) ,OTU(p29r16.fault_ack.6) ];
   87: NEQ(p29r16.fault,p29r16.fault_ack)OTE(p29r16.unack_fault);
   // Warnings
   88: OTE(p29r16.comment.31);
   89: XIC(p01r09_pb_global_reset)MOV(p29r16.warning,p29r16.warning_ack);
   90: XIC(p29_wdb_status_word.7)[TON(p29r16_timer_warning[0],?,?) ,XIC(p29r16_timer_warning[0].DN) OTL(p29r16.warning.0) ];
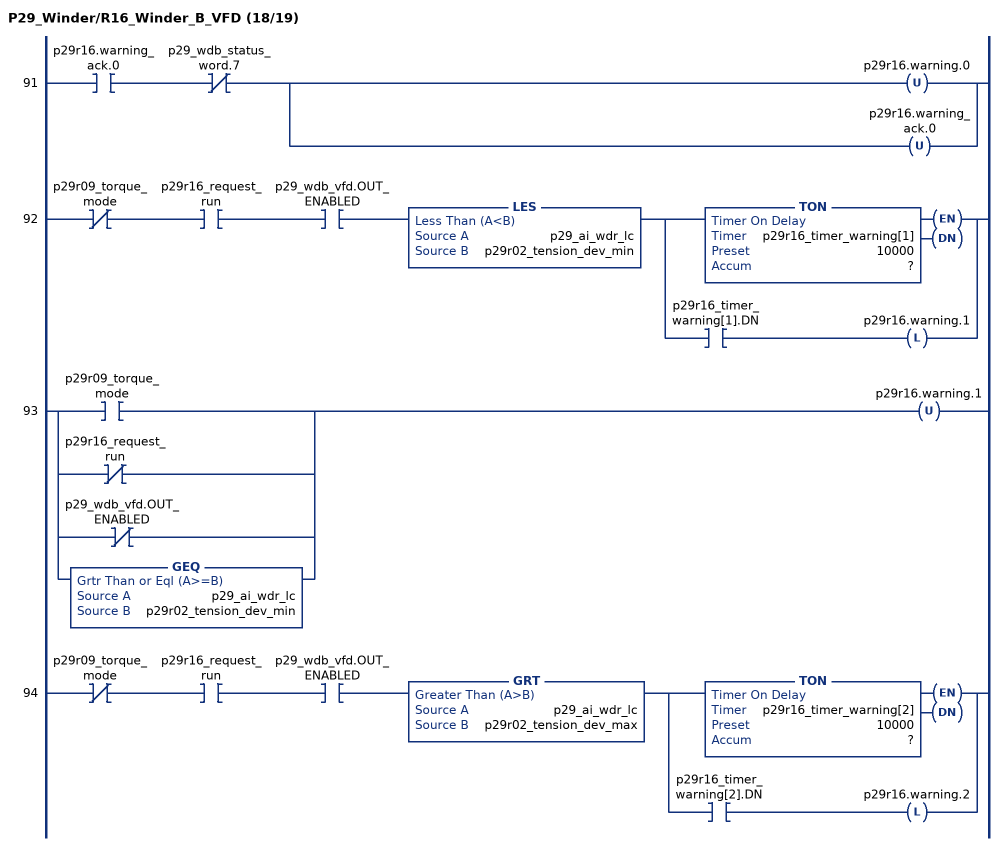
   91: XIC(p29r16.warning_ack.0)XIO(p29_wdb_status_word.7)[OTU(p29r16.warning.0) ,OTU(p29r16.warning_ack.0) ];
   92: XIO(p29r09_torque_mode)XIC(p29r16_request_run)XIC(p29_wdb_vfd.OUT_ENABLED)LES(p29_ai_wdr_lc,p29r02_tension_dev_min)[TON(p29r16_timer_warning[1],?,?) ,XIC(p29r16_timer_warning[1].DN) OTL(p29r16.warning.1) ];
   93: [XIC(p29r09_torque_mode) ,XIO(p29r16_request_run) ,XIO(p29_wdb_vfd.OUT_ENABLED) ,GEQ(p29_ai_wdr_lc,p29r02_tension_dev_min) ]OTU(p29r16.warning.1);
   94: XIO(p29r09_torque_mode)XIC(p29r16_request_run)XIC(p29_wdb_vfd.OUT_ENABLED)GRT(p29_ai_wdr_lc,p29r02_tension_dev_max)[TON(p29r16_timer_warning[2],?,?) ,XIC(p29r16_timer_warning[2].DN) OTL(p29r16.warning.2) ];
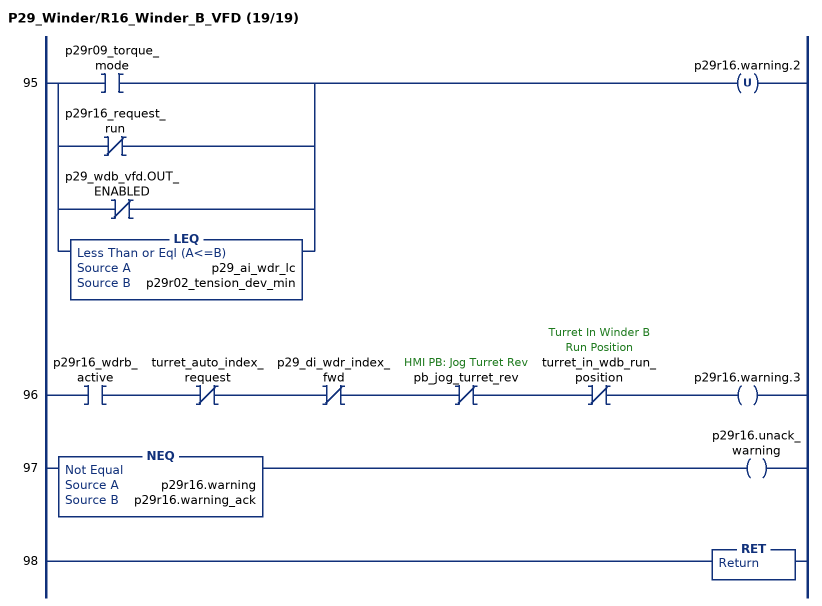
   95: [XIC(p29r09_torque_mode) ,XIO(p29r16_request_run) ,XIO(p29_wdb_vfd.OUT_ENABLED) ,LEQ(p29_ai_wdr_lc,p29r02_tension_dev_min) ]OTU(p29r16.warning.2);
   96: XIC(p29r16_wdrb_active)XIO(turret_auto_index_request)XIO(p29_di_wdr_index_fwd)XIO(pb_jog_turret_rev)XIO(turret_in_wdb_run_position)OTE(p29r16.warning.3);
   97: NEQ(p29r16.warning,p29r16.warning_ack)OTE(p29r16.unack_warning);
   98: RET();
END_ROUTINE
